(* IEC 61131-3 sources: windowtracking/src/Items, 2 files *)

(* ---- IItem.st ---- *)
USING Simatic.Ax.WindowTracking;

NAMESPACE Simatic.Ax.WindowTracking
    INTERFACE IItem
        METHOD GetDestination : IVirtualTrigger
            VAR_INPUT
                id : UINT;
            END_VAR
        END_METHOD
        METHOD DestinationCount : INT
        END_METHOD
    END_INTERFACE
END_NAMESPACE

(* ---- Item1Destination.st ---- *)
NAMESPACE Simatic.Ax.WindowTracking
    CLASS ItemOneDestination IMPLEMENTS IItem

        VAR PUBLIC
            Destination1 : IVirtualTrigger;
        END_VAR

        METHOD PUBLIC GetDestination : IVirtualTrigger
            VAR_INPUT
                id : UINT := UINT#0;
            END_VAR
            GetDestination := Destination1;
        END_METHOD

        METHOD PUBLIC DestinationCount : INT
            IF (Destination1 <> NULL) THEN
                DestinationCount := 1;
            ELSE
                DestinationCount := 0;
            END_IF;
        END_METHOD
    END_CLASS
END_NAMESPACE
